FUNCTION_BLOCK CalculatePosAngle
VAR_INPUT
	X1			: LREAL;
	X2			: LREAL;
	Y1			: LREAL;
	Y2			: LREAL;
END_VAR
VAR_OUTPUT
	alrResult		: ARRAY[0..2] OF LREAL;
END_VAR
VAR
END_VAR

alrResult[0] := X1;
alrResult[1] := Y1;
alrResult[2] := RAD_TO_DEG(ATAN((Y2-Y1)/(X2-X1)));

END_FUNCTION_BLOCK

(* stored: Version 1.1.0.1, ProductVersion 3.1.4022.12
   POU CalculatePosAngle: Id {2a22d496-cc99-4e1b-8eeb-c65ce7ebc0f1}, SpecialFunc None *)
